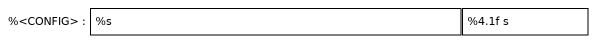
[picture p205: ZLIB_SFC_STATE (HMI screen)]
rectangle at (0,0)-(231,27): text "%<CONFIG> :"; shows $SFC$.SFCCurrentPOU
rectangle at (230,0)-(601,27): text "%s"; shows $SFC$.SFCCurrentStep
rectangle at (602,0)-(728,27): text "%4.1f s"; shows $SFC$.SFCTime / 1000.0
*)

(* Visualisation zLibrary/MessageHandler/ZLIB_SHOWMESSAGEBUTTON
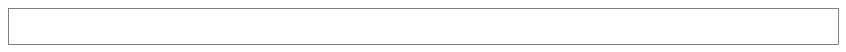
polyline at (830,0)-(830,36): invisible if NOT $Object$.Visible; alarm colour if $Object$.Pressed
polyline at (0,36)-(830,36): invisible if NOT $Object$.Visible; alarm colour if $Object$.Pressed
polyline at (6,0)-(823,0): invisible if NOT $Object$.Visible; alarm colour if NOT $Object$.Pressed
polyline at (0,0)-(0,36): invisible if NOT $Object$.Visible; alarm colour if NOT $Object$.Pressed
polyline at (0,36)-(830,36): invisible if NOT $Object$.Visible; alarm colour if $Object$.Pressed
polyline at (830,0)-(830,36): invisible if NOT $Object$.Visible; alarm colour if $Object$.Pressed
polyline at (0,0)-(830,0): invisible if NOT $Object$.Visible; alarm colour if NOT $Object$.Pressed
polyline at (0,0)-(0,36): invisible if NOT $Object$.Visible; alarm colour if NOT $Object$.Pressed
1 elements of other kinds (tables, trends, ...) not read
*)

(* Visualisation zLibrary/ept/TippiDrucker/ZLIB_TIPPL
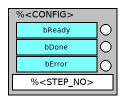
rectangle at (0,0)-(109,87): text "%<CONFIG>"; shows '$Objekt$'
rectangle at (5,27)-(87,46): text "%<BASIC>"; shows 'bDone'
rectangle at (5,47)-(87,66): text "%<BASIC>"; shows 'bError'
ellipse at (92,33)-(103,44): alarm colour if $Objekt$.bDone
ellipse at (92,52)-(103,63): alarm colour if $Objekt$.bError
ellipse at (92,16)-(103,27): alarm colour if $Objekt$.bReady
rectangle at (5,12)-(88,31): text "%<BASIC>"; shows 'bReady'
rectangle at (8,14)-(89,30): text "bReady"; invisible if TRUE
rectangle at (8,31)-(89,47): text "bDone"; invisible if TRUE
rectangle at (8,48)-(89,64): text "bError"; invisible if TRUE
rectangle at (4,66)-(105,82): text "%<STEP_NO>"; shows $Objekt$.fb_state_entry.i16_step; alarm colour if $Objekt$.fb_state_entry.i16_step = FEHLER
rectangle at (4,66)-(105,82): text "%<STEP_NO>"; shows $Objekt$.fb_state_entry.i16_step; invisible if $Objekt$.fb_state_entry.i16_step >= 980; alarm colour if $Objekt$.fb_state_entry.i16_step = 100
*)

(* Visualisation zLibrary/Valve/ZLIB_VALVE_1_SENSORS
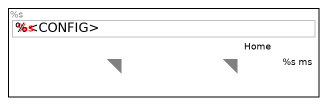
rectangle at (0,0)-(311,89): text "%s"; shows $Object$.BitName
rectangle at (5,11)-(306,28): text "%<CONFIG>"; shows $Object$.InstName
rounded rectangle at (234,32)-(280,45): text "Home"; shows $Object$.State
rectangle at (235,46)-(306,62): text "%s ms"; shows $Object$.ProcessTime
rounded rectangle at (4,12)-(307,29): text "%s"; shows $Object$.ErrorString; invisible if NOT $Object$.ErrorPresent
polygon at (99,51)-(113,65): invisible if $Object$.NoOfValveCoils<2; alarm colour if $Object$.CoilB
polygon at (215,51)-(229,65): alarm colour if $Object$.CoilA
6 elements of other kinds (tables, trends, ...) not read
*)

(* Visualisation zLibrary/Valve/ZLIB_VALVE_2_SENSORS
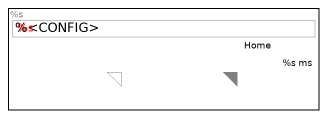
rectangle at (0,0)-(311,102): text "%s"; shows $Object$.BitName
rounded rectangle at (234,31)-(280,44): text "Home"; shows $Object$.State
rectangle at (235,47)-(306,63): text "%s ms"; shows $Object$.ProcessTime
rectangle at (5,11)-(306,28): text "%<CONFIG>"; shows $Object$.InstName
rounded rectangle at (4,12)-(307,29): text "%s"; shows $Object$.ErrorString; invisible if NOT $Object$.ErrorPresent
polygon at (99,64)-(113,78): invisible if $Object$.NoOfValveCoils<2; alarm colour if $Object$.CoilB
polygon at (215,64)-(229,78): alarm colour if $Object$.CoilA
8 elements of other kinds (tables, trends, ...) not read
*)

(* Visualisation zLibrary/Valve/ZLIB_VALVE_3_SENSORS
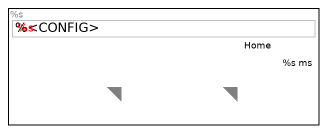
rectangle at (0,0)-(311,117): text "%s"; shows $Object$.BitName
rounded rectangle at (234,31)-(280,44): text "Home"; shows $Object$.State
rectangle at (235,47)-(306,63): text "%s ms"; shows $Object$.ProcessTime
rectangle at (5,11)-(306,28): text "%<CONFIG>"; shows $Object$.InstName
rounded rectangle at (4,12)-(307,29): text "%s"; shows $Object$.ErrorString; invisible if NOT $Object$.ErrorPresent
polygon at (99,79)-(113,93): invisible if $Object$.NoOfValveCoils<2; alarm colour if $Object$.CoilB
polygon at (215,79)-(229,93): alarm colour if $Object$.CoilA
10 elements of other kinds (tables, trends, ...) not read
*)

(* Visualisation zLibrary/Valve/ZLIB_VALVE_5_SENSORS
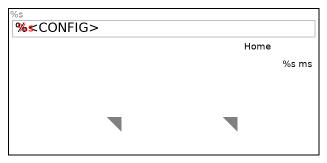
rectangle at (0,0)-(311,147): text "%s"; shows $Object$.BitName
rounded rectangle at (234,32)-(280,45): text "Home"; shows $Object$.State
rectangle at (235,48)-(306,64): text "%s ms"; shows $Object$.ProcessTime
rectangle at (5,11)-(306,28): text "%<CONFIG>"; shows $Object$.InstName
rounded rectangle at (4,12)-(307,29): text "%s"; shows $Object$.ErrorString; invisible if NOT $Object$.ErrorPresent
polygon at (99,109)-(113,123): invisible if $Object$.NoOfValveCoils<2; alarm colour if $Object$.CoilB
polygon at (215,109)-(229,123): alarm colour if $Object$.CoilA
14 elements of other kinds (tables, trends, ...) not read
*)

(* Visualisation zLibrary/VisuObjects/ZLIB_VISUBUTTON
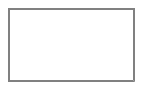
polyline at (125,1)-(125,72): invisible if NOT $Object$.Visible; alarm colour if $Object$.Pressed
polyline at (1,72)-(125,72): invisible if NOT $Object$.Visible; alarm colour if $Object$.Pressed
polyline at (1,1)-(125,1): invisible if NOT $Object$.Visible; alarm colour if NOT $Object$.Pressed
polyline at (1,1)-(1,72): invisible if NOT $Object$.Visible; alarm colour if NOT $Object$.Pressed
polyline at (0,73)-(126,73): invisible if NOT $Object$.Visible; alarm colour if $Object$.Pressed
polyline at (126,0)-(126,73): invisible if NOT $Object$.Visible; alarm colour if $Object$.Pressed
polyline at (0,0)-(126,0): invisible if NOT $Object$.Visible; alarm colour if NOT $Object$.Pressed
polyline at (0,0)-(0,73): invisible if NOT $Object$.Visible; alarm colour if NOT $Object$.Pressed
1 elements of other kinds (tables, trends, ...) not read
*)

(* Visualisation zLibrary/VisuObjects/ZLIB_VISUBUTTON_ARROW_DOWN
1 elements of other kinds (tables, trends, ...) not read
*)

(* Visualisation zLibrary/VisuObjects/ZLIB_VISUBUTTON_ARROW_UP
1 elements of other kinds (tables, trends, ...) not read
*)

(* Visualisation zLibrary/VisuObjects/ZLIB_VISUBUTTON_MODE_SELECT
1 elements of other kinds (tables, trends, ...) not read
*)

(* Visualisation zLibrary/VisuObjects/ZLIB_VISUBUTTON_S17
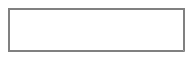
polyline at (175,1)-(175,42): invisible if NOT $Object$.Visible; alarm colour if $Object$.Pressed
polyline at (1,42)-(175,42): invisible if NOT $Object$.Visible; alarm colour if $Object$.Pressed
polyline at (1,1)-(175,1): invisible if NOT $Object$.Visible; alarm colour if NOT $Object$.Pressed
polyline at (1,1)-(1,42): invisible if NOT $Object$.Visible; alarm colour if NOT $Object$.Pressed
polyline at (0,43)-(176,43): invisible if NOT $Object$.Visible; alarm colour if $Object$.Pressed
polyline at (176,0)-(176,43): invisible if NOT $Object$.Visible; alarm colour if $Object$.Pressed
polyline at (0,0)-(176,0): invisible if NOT $Object$.Visible; alarm colour if NOT $Object$.Pressed
polyline at (0,0)-(0,43): invisible if NOT $Object$.Visible; alarm colour if NOT $Object$.Pressed
1 elements of other kinds (tables, trends, ...) not read
*)

(* Visualisation zLibrary/VisuObjects/ZLIB_VISUBUTTON_S18
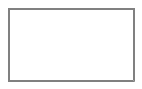
polyline at (125,1)-(125,72): invisible if NOT $Object$.Visible; alarm colour if $Object$.Pressed
polyline at (1,72)-(125,72): invisible if NOT $Object$.Visible; alarm colour if $Object$.Pressed
polyline at (1,1)-(125,1): invisible if NOT $Object$.Visible; alarm colour if NOT $Object$.Pressed
polyline at (1,1)-(1,72): invisible if NOT $Object$.Visible; alarm colour if NOT $Object$.Pressed
polyline at (0,73)-(126,73): invisible if NOT $Object$.Visible; alarm colour if $Object$.Pressed
polyline at (126,0)-(126,73): invisible if NOT $Object$.Visible; alarm colour if $Object$.Pressed
polyline at (0,0)-(126,0): invisible if NOT $Object$.Visible; alarm colour if NOT $Object$.Pressed
polyline at (0,0)-(0,73): invisible if NOT $Object$.Visible; alarm colour if NOT $Object$.Pressed
1 elements of other kinds (tables, trends, ...) not read
*)

(* Visualisation zLibrary/VisuObjects/ZLIB_VISUBUTTON_S24
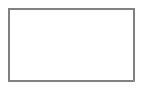
polyline at (125,1)-(125,72): invisible if NOT $Object$.Visible; alarm colour if $Object$.Pressed
polyline at (1,72)-(125,72): invisible if NOT $Object$.Visible; alarm colour if $Object$.Pressed
polyline at (1,1)-(125,1): invisible if NOT $Object$.Visible; alarm colour if NOT $Object$.Pressed
polyline at (1,1)-(1,72): invisible if NOT $Object$.Visible; alarm colour if NOT $Object$.Pressed
polyline at (0,73)-(126,73): invisible if NOT $Object$.Visible; alarm colour if $Object$.Pressed
polyline at (126,0)-(126,73): invisible if NOT $Object$.Visible; alarm colour if $Object$.Pressed
polyline at (0,0)-(126,0): invisible if NOT $Object$.Visible; alarm colour if NOT $Object$.Pressed
polyline at (0,0)-(0,73): invisible if NOT $Object$.Visible; alarm colour if NOT $Object$.Pressed
1 elements of other kinds (tables, trends, ...) not read
*)

(* Visualisation zLibrary/VisuObjects/ZLIB_VISUBUTTON_S24_S
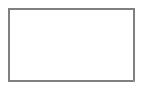
polyline at (125,1)-(125,72): invisible if NOT $Object$.Visible; alarm colour if $Object$.Pressed
polyline at (1,72)-(125,72): invisible if NOT $Object$.Visible; alarm colour if $Object$.Pressed
polyline at (1,1)-(125,1): invisible if NOT $Object$.Visible; alarm colour if NOT $Object$.Pressed
polyline at (1,1)-(1,72): invisible if NOT $Object$.Visible; alarm colour if NOT $Object$.Pressed
polyline at (0,73)-(126,73): invisible if NOT $Object$.Visible; alarm colour if $Object$.Pressed
polyline at (126,0)-(126,73): invisible if NOT $Object$.Visible; alarm colour if $Object$.Pressed
polyline at (0,0)-(126,0): invisible if NOT $Object$.Visible; alarm colour if NOT $Object$.Pressed
polyline at (0,0)-(0,73): invisible if NOT $Object$.Visible; alarm colour if NOT $Object$.Pressed
1 elements of other kinds (tables, trends, ...) not read
*)

(* Visualisation zLibrary/VisuObjects/ZLIB_VISUBUTTON_S24_S_IO
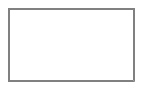
polyline at (125,1)-(125,72): invisible if NOT $Object$.Visible; alarm colour if $Object$.Pressed
polyline at (1,72)-(125,72): invisible if NOT $Object$.Visible; alarm colour if $Object$.Pressed
polyline at (1,1)-(125,1): invisible if NOT $Object$.Visible; alarm colour if NOT $Object$.Pressed
polyline at (1,1)-(1,72): invisible if NOT $Object$.Visible; alarm colour if NOT $Object$.Pressed
polyline at (0,73)-(126,73): invisible if NOT $Object$.Visible; alarm colour if $Object$.Pressed
polyline at (126,0)-(126,73): invisible if NOT $Object$.Visible; alarm colour if $Object$.Pressed
polyline at (0,0)-(126,0): invisible if NOT $Object$.Visible; alarm colour if NOT $Object$.Pressed
polyline at (0,0)-(0,73): invisible if NOT $Object$.Visible; alarm colour if NOT $Object$.Pressed
1 elements of other kinds (tables, trends, ...) not read
*)

(* Visualisation zLibrary/VisuObjects/ZLIB_VISUBUTTON_S36
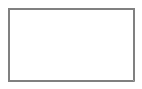
polyline at (125,1)-(125,72): invisible if NOT $Object$.Visible; alarm colour if $Object$.Pressed
polyline at (1,72)-(125,72): invisible if NOT $Object$.Visible; alarm colour if $Object$.Pressed
polyline at (1,1)-(125,1): invisible if NOT $Object$.Visible; alarm colour if NOT $Object$.Pressed
polyline at (1,1)-(1,72): invisible if NOT $Object$.Visible; alarm colour if NOT $Object$.Pressed
polyline at (0,73)-(126,73): invisible if NOT $Object$.Visible; alarm colour if $Object$.Pressed
polyline at (126,0)-(126,73): invisible if NOT $Object$.Visible; alarm colour if $Object$.Pressed
polyline at (0,0)-(126,0): invisible if NOT $Object$.Visible; alarm colour if NOT $Object$.Pressed
polyline at (0,0)-(0,73): invisible if NOT $Object$.Visible; alarm colour if NOT $Object$.Pressed
1 elements of other kinds (tables, trends, ...) not read
*)

(* Visualisation zLibrary/VisuObjects/SERVICE/ZLIB_VISUBUTTON_TOGGELN
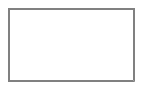
polyline at (125,1)-(125,72): invisible if NOT $Object$.Visible; alarm colour if $Object$.Pressed
polyline at (1,72)-(125,72): invisible if NOT $Object$.Visible; alarm colour if $Object$.Pressed
polyline at (1,1)-(125,1): invisible if NOT $Object$.Visible; alarm colour if NOT $Object$.Pressed
polyline at (1,1)-(1,72): invisible if NOT $Object$.Visible; alarm colour if NOT $Object$.Pressed
polyline at (0,73)-(126,73): invisible if NOT $Object$.Visible; alarm colour if $Object$.Pressed
polyline at (126,0)-(126,73): invisible if NOT $Object$.Visible; alarm colour if $Object$.Pressed
polyline at (0,0)-(126,0): invisible if NOT $Object$.Visible; alarm colour if NOT $Object$.Pressed
polyline at (0,0)-(0,73): invisible if NOT $Object$.Visible; alarm colour if NOT $Object$.Pressed
1 elements of other kinds (tables, trends, ...) not read
*)

(* Visualisation zLibrary/MessageHandler/ZLIB_VISUMESSAGEHANDLER
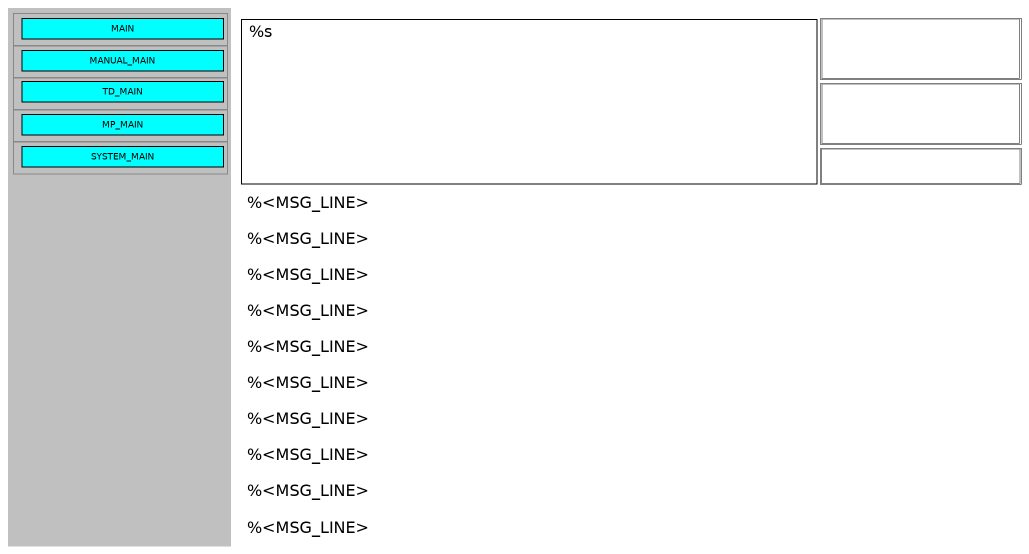
embedded screen at (815,190)-(1016,251): ZLIB_VISUBUTTON
embedded screen at (815,255)-(1016,291): ZLIB_VISUBUTTON_S17
embedded screen at (235,295)-(1014,324): zLib_MessageLine
embedded screen at (235,331)-(1016,360): zLib_MessageLine
embedded screen at (235,367)-(1016,396): zLib_MessageLine
embedded screen at (235,403)-(1016,432): zLib_MessageLine
embedded screen at (235,439)-(1016,468): zLib_MessageLine
embedded screen at (235,475)-(1016,504): zLib_MessageLine
embedded screen at (235,511)-(1016,540): zLib_MessageLine
embedded screen at (235,547)-(1016,576): zLib_MessageLine
embedded screen at (235,583)-(1016,612): zLib_MessageLine
embedded screen at (235,620)-(1016,649): zLib_MessageLine
embedded screen at (815,125)-(1016,186): ZLIB_VISUBUTTON
embedded screen at (3,115)-(226,653): M0000_Main
rectangle at (242,128)-(808,289): text "%s"; shows .Visu.Message.Text
1 more shapes without text or variables
1 elements of other kinds (tables, trends, ...) not read
*)

(* Visualisation zLibrary/VisuObjects/ZLIBVISUBUTTON_TEXTINPUT
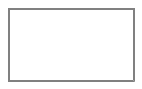
polyline at (125,1)-(125,72): invisible if NOT $Object$.Visible; alarm colour if $Object$.Pressed
polyline at (1,72)-(125,72): invisible if NOT $Object$.Visible; alarm colour if $Object$.Pressed
polyline at (1,1)-(125,1): invisible if NOT $Object$.Visible; alarm colour if NOT $Object$.Pressed
polyline at (1,1)-(1,72): invisible if NOT $Object$.Visible; alarm colour if NOT $Object$.Pressed
polyline at (0,73)-(126,73): invisible if NOT $Object$.Visible; alarm colour if $Object$.Pressed
polyline at (126,0)-(126,73): invisible if NOT $Object$.Visible; alarm colour if $Object$.Pressed
polyline at (0,0)-(126,0): invisible if NOT $Object$.Visible; alarm colour if NOT $Object$.Pressed
polyline at (0,0)-(0,73): invisible if NOT $Object$.Visible; alarm colour if NOT $Object$.Pressed
1 elements of other kinds (tables, trends, ...) not read
*)

(* Visualisation zLibrary/VisuObjects/ZLIBVISUBUTTON_TEXTVAR
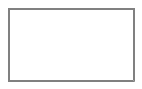
polyline at (125,1)-(125,72): invisible if NOT $Object$.Visible; alarm colour if $Object$.Pressed
polyline at (1,72)-(125,72): invisible if NOT $Object$.Visible; alarm colour if $Object$.Pressed
polyline at (1,1)-(125,1): invisible if NOT $Object$.Visible; alarm colour if NOT $Object$.Pressed
polyline at (1,1)-(1,72): invisible if NOT $Object$.Visible; alarm colour if NOT $Object$.Pressed
polyline at (0,73)-(126,73): invisible if NOT $Object$.Visible; alarm colour if $Object$.Pressed
polyline at (126,0)-(126,73): invisible if NOT $Object$.Visible; alarm colour if $Object$.Pressed
polyline at (0,0)-(126,0): invisible if NOT $Object$.Visible; alarm colour if NOT $Object$.Pressed
polyline at (0,0)-(0,73): invisible if NOT $Object$.Visible; alarm colour if NOT $Object$.Pressed
1 elements of other kinds (tables, trends, ...) not read
*)

(* Visualisation zLibrary/VisuObjects/ZLIBVISUBUTTON_ZOOMTOCALLER
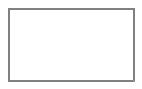
polyline at (125,1)-(125,72): invisible if NOT $Object$.Visible; alarm colour if $Object$.Pressed
polyline at (1,72)-(125,72): invisible if NOT $Object$.Visible; alarm colour if $Object$.Pressed
polyline at (1,1)-(125,1): invisible if NOT $Object$.Visible; alarm colour if NOT $Object$.Pressed
polyline at (1,1)-(1,72): invisible if NOT $Object$.Visible; alarm colour if NOT $Object$.Pressed
polyline at (0,73)-(126,73): invisible if NOT $Object$.Visible; alarm colour if $Object$.Pressed
polyline at (126,0)-(126,73): invisible if NOT $Object$.Visible; alarm colour if $Object$.Pressed
polyline at (0,0)-(126,0): invisible if NOT $Object$.Visible; alarm colour if NOT $Object$.Pressed
polyline at (0,0)-(0,73): invisible if NOT $Object$.Visible; alarm colour if NOT $Object$.Pressed
1 elements of other kinds (tables, trends, ...) not read
*)

(* Visualisation zLibrary/ept/Zuführungen/ZUFUEHRUNG
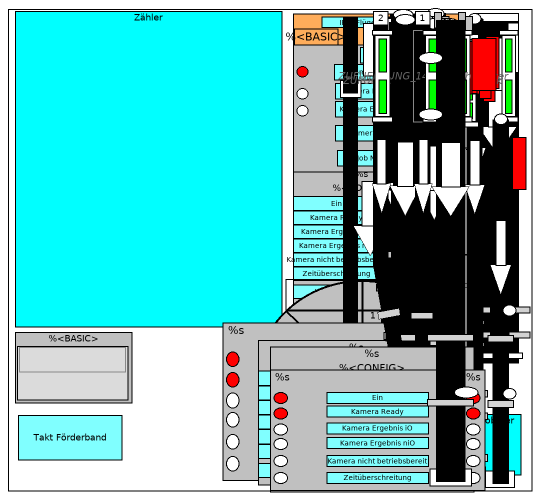
group at (0,1)-(524,483)
  rectangle at (0,0)-(524,482): invisible if TRUE
  rectangle at (464,405)-(513,466): text "Roboter"; invisible if TRUE; opens MANUAL_ST03_0
  rectangle at (7,2)-(274,318): text "Zähler"; invisible if TRUE; opens MANUAL_ST03_0
rectangle at (10,407)-(114,452): text "Takt Förderband"; invisible if TRUE
rectangle at (7,324)-(124,395): text "%<BASIC>"; shows 'Föderband'; invisible if MP.ST03.SGM_3621
embedded screen at (9,338)-(120,392): ZLIB_OVERRIDE
embedded screen at (245,5)-(522,481): ZUFUEHRUNG_93POL
embedded screen at (360,1)-(423,473): ZUFUEHRUNG_92POL
embedded screen at (331,9)-(392,480): ZUFUEHRUNG_154RP
embedded screen at (423,7)-(464,483): ZUFUEHRUNG_74_91_168POL
embedded screen at (378,8)-(419,480): ZUFUEHRUNG_154POL
embedded screen at (400,0)-(460,481): ZUFUEHRUNG_35POL
embedded screen at (348,5)-(420,477): ZUFUEHRUNG_206POL
embedded screen at (368,2)-(440,474): ZUFUEHRUNG_124POL
embedded screen at (332,3)-(483,475): ZUFUEHRUNG_46POL
embedded screen at (142,6)-(496,473): ZUFUEHRUNG_NOX_5_6POL
embedded screen at (250,5)-(491,477): ZUFUEHRUNG_NOX_4POL
embedded screen at (390,8)-(462,480): ZUFUEHRUNG_88POL
embedded screen at (394,7)-(487,478): ZUFUEHRUNG_7POL
embedded screen at (409,10)-(479,482): ZUFUEHRUNG_88POL_AMG
embedded screen at (404,10)-(474,482): ZUFUEHRUNG_120POL
embedded screen at (399,10)-(469,482): ZUFUEHRUNG_21POL
embedded screen at (394,10)-(464,482): ZUFUEHRUNG_191POL
embedded screen at (363,1)-(433,477): ZUFUEHRUNG_72POL
embedded screen at (365,6)-(435,477): ZUFUEHRUNG_48POL
embedded screen at (328,3)-(510,479): ZUFUEHRUNG_268POL_RP
embedded screen at (262,7)-(518,484): ZUFUEHRUNG_268POL_102POL_NEU
embedded screen at (404,7)-(488,478): ZUFUEHRUNG_33POL
1 elements of other kinds (tables, trends, ...) not read
*)

(* Visualisation zLibrary/ept/Zuführungen/ZUFUEHRUNG_120POL
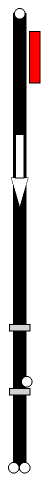
embedded screen at (9,126)-(26,199): SIGNS_ARROWDOWN
ellipse at (12,0)-(23,11): alarm colour if ST03_531_B69_0.BitInToCheck; tooltip ST03_531_B69_0
ellipse at (19,368)-(30,379): alarm colour if ST03_531_B69_6.BitInToCheck; tooltip ST03_531_B69_6
rectangle at (7,380)-(28,387): alarm colour if ST03_531_B69_4.ValveSensor; tooltip ST03_531_B69_3
rectangle at (7,316)-(28,323): alarm colour if ST03_531_B69_2.ValveSensor; tooltip ST03_531_B69_1
rounded rectangle at (27,23)-(38,75): alarm colour if ST03_Init_Lockings.b_freiFuerSG; tooltip b_freiFuerSG
ellipse at (17,454)-(28,465): alarm colour if ST03_531_B69_7.BitInToCheck; tooltip ST03_531_B69_7
ellipse at (6,454)-(17,465): alarm colour if ST03_532_B70_0.BitInToCheck; tooltip ST03_532_B70_0
2 more shapes without text or variables
*)

(* Visualisation zLibrary/ept/Zuführungen/ZUFUEHRUNG_124POL
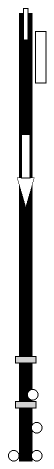
ellipse at (10,447)-(21,458): alarm colour if ST03_452_B70_1.BitInToCheck; tooltip ST03_452_B70_1
embedded screen at (19,131)-(36,204): SIGNS_ARROWDOWN
ellipse at (33,419)-(44,430): alarm colour if ST03_452_B70_2.BitInToCheck; tooltip ST03_452_B70_2
ellipse at (33,447)-(44,458): alarm colour if ST03_453_B70_4.BitInToCheck; tooltip ST03_453_B70_4
ellipse at (29,386)-(40,397): alarm colour if ST03_451_B69_7.BitInToCheck; tooltip ST03_451_B69_7
rectangle at (17,398)-(38,405): alarm colour if ST03_451_B69_2.ValveSensor; tooltip ST03_451_B69_2
rectangle at (17,353)-(38,360): alarm colour if ST03_451_B69_1.ValveSensor; tooltip ST03_451_B69_1
rounded rectangle at (37,28)-(48,80): alarm colour if ST03_Init_Lockings.b_freiFuerSG; tooltip b_freiFuerSG
rounded rectangle at (25,5)-(30,37): alarm colour if ST03_451_B69_4.BitInToCheck; tooltip ST03_451_B69_4
1 more shapes without text or variables
*)

(* Visualisation zLibrary/ept/Zuführungen/ZUFUEHRUNG_154POL
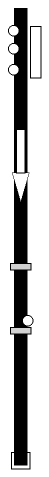
ellipse at (5,35)-(16,46): alarm colour if ST03_425_B67_5.BitInToCheck; tooltip ST03_425_B67_5
embedded screen at (9,121)-(26,194): SIGNS_ARROWDOWN
ellipse at (5,56)-(16,67): alarm colour if ST03_425_B67_6.BitInToCheck; tooltip ST03_425_B67_6
ellipse at (5,17)-(16,28): alarm colour if ST03_425_B67_4.BitInToCheck; tooltip ST03_425_B67_4
ellipse at (19,307)-(30,318): alarm colour if ST03_425_B67_7.BitInToCheck; tooltip ST03_425_B67_7
rectangle at (7,319)-(28,326): alarm colour if ST03_425_B67_2.ValveSensor; tooltip ST03_425_B67_2
rectangle at (7,255)-(28,262): alarm colour if ST03_425_B67_0.ValveSensor; tooltip ST03_425_B67_0
rounded rectangle at (8,444)-(27,461): alarm colour if ST03_426_B68_4.BitInToCheck; tooltip ST03_426_B68_4
rounded rectangle at (27,18)-(38,70): alarm colour if ST03_Init_Lockings.b_freiFuerSG; tooltip b_freiFuerSG
2 more shapes without text or variables
*)

(* Visualisation zLibrary/ept/Zuführungen/ZUFUEHRUNG_154RP
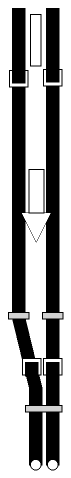
embedded screen at (13,161)-(43,234): SIGNS_ARROWDOWN
ellipse at (39,451)-(50,462): alarm colour if ST03_419_B61_3.BitInToCheck; tooltip ST03_419_B61_3
ellipse at (22,451)-(33,462): alarm colour if ST03_419_B61_2.BitInToCheck; tooltip ST03_419_B61_2
rounded rectangle at (35,350)-(54,367): alarm colour if ST03_419_B61_1.BitInToCheck; tooltip ST03_419_B61_1
rounded rectangle at (14,350)-(33,367): alarm colour if ST03_419_B61_0.BitInToCheck; tooltip ST03_419_B61_0
rectangle at (17,397)-(54,404): alarm colour if ST03_418_B60_5.ValveSensor; tooltip ST03_418_B60_5
rectangle at (0,304)-(21,311): alarm colour if ST03_418_B60_0.ValveSensor; tooltip ST03_418_B60_0
rectangle at (34,304)-(55,311): alarm colour if ST03_418_B60_2.ValveSensor; tooltip ST03_418_B60_2
rounded rectangle at (35,61)-(54,78): alarm colour if ST03_418_B60_7.BitInToCheck; tooltip ST03_418_B60_7
rounded rectangle at (1,62)-(20,79): alarm colour if ST03_418_B60_6.BitInToCheck; tooltip ST03_418_B60_6
rounded rectangle at (22,6)-(33,58): alarm colour if ST03_Init_Lockings.b_freiFuerSG; tooltip b_freiFuerSG
8 more shapes without text or variables
*)

(* Visualisation zLibrary/ept/Zuführungen/ZUFUEHRUNG_160POL
